ABB RobotStudio station: L4_1_20220629-155623.rsstn

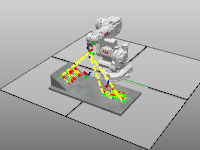
Station L4_1 (saved by RobotStudio 20.4.9280.0)
Controller IRB140_6_81
  mechanical unit ROB_1: IRB140_6_81_C_03, 6 joints, base frame (0, 0, 0) mm
Layout (positions relative to the parent item):
  - IRB140_6_81_C_03 [mechanism, from Robots\IRB140_6_81_C_G_03.rslib] at (0, 0, 0) mm; joint values [0, 0, 0, 0, 0.5236, 0] (rad or m)
  - MyNewTool [mechanism] at (506.29, 0, 679.5) mm, rotated rx 180 ry 60 rz 180 deg
      TCP Point at (78.44, 0, 73.52) mm, rotated rx 0 ry 70 rz 0 deg
      links: Tool
  - BaseBoard [part]
  - InclinedBoard [part] at (230, -500, 30) mm
Attachment: MyNewTool is attached to IRB140_6_81_C_03 / Link6
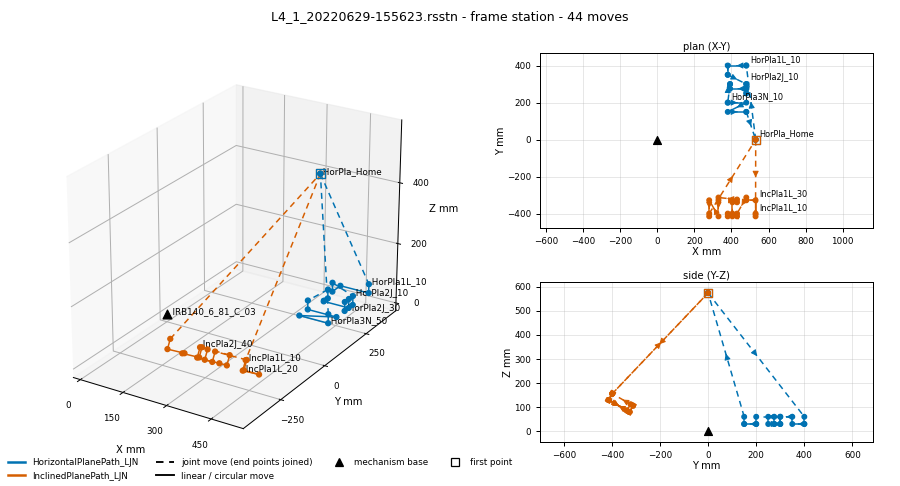
[picture p0: tool path of L4_1_20220629-155623.rsstn in frame station, 44 of 44 moves have a stored position in this frame; points joined in program order, loops and branches not executed]
Targets, tools, work objects and paths stored in the station, written as RAPID:
! task T_ROB1
MODULE CalibData
  TASK PERS wobjdata WO_InclinedPlane:=[FALSE,TRUE,"",[[230,-240.192,30],[0.68301276,-0.183012486,-0.183012486,-0.68301276]],[[0,0,30],[1,0,0,0]]];
  PERS tooldata Point:=[TRUE,[[78.437,0,73.516],[0.819152044,0,0.573576436,0]],[0.25,[0,0,1],[1,0,0,0],0,0,0]];
  TASK PERS wobjdata WO_HorizontalPlane:=[FALSE,TRUE,"",[[280,100,30],[1,0,0,0]],[[0,0,30],[1,0,0,0]]];
ENDMODULE

! task T_ROB1
MODULE Module1
  CONST robtarget HorPla2J_20:=[[200,200,-30],[0,0,1,0],[0,0,-1,1],[9E+09,9E+09,9E+09,9E+09,9E+09,9E+09]];
  CONST robtarget HorPla2J_10:=[[200,200,0],[0,0,1,0],[0,0,-1,1],[9E+09,9E+09,9E+09,9E+09,9E+09,9E+09]];
  CONST robtarget HorPla2J_30:=[[200,150,-30],[0,0,1,0],[0,0,-1,1],[9E+09,9E+09,9E+09,9E+09,9E+09,9E+09]];
  CONST robtarget HorPla2J_40:=[[200,150,0],[0,0,1,0],[0,0,-1,1],[9E+09,9E+09,9E+09,9E+09,9E+09,9E+09]];
  CONST robtarget HorPla2J_60:=[[200,175,-30],[0,0,1,0],[0,0,-1,1],[9E+09,9E+09,9E+09,9E+09,9E+09,9E+09]];
  CONST robtarget HorPla2J_50:=[[200,175,0],[0,0,1,0],[0,0,-1,1],[9E+09,9E+09,9E+09,9E+09,9E+09,9E+09]];
  CONST robtarget HorPla2J_70:=[[112.5,175,-30],[0,0,1,0],[0,0,-1,1],[9E+09,9E+09,9E+09,9E+09,9E+09,9E+09]];
  CONST robtarget HorPla2J_80:=[[100,187.5,-30],[0,0,1,0],[0,0,0,1],[9E+09,9E+09,9E+09,9E+09,9E+09,9E+09]];
  CONST robtarget HorPla2J_90:=[[112.5,200,-30],[0,0,1,0],[0,0,-1,1],[9E+09,9E+09,9E+09,9E+09,9E+09,9E+09]];
  CONST robtarget HorPla2J_100:=[[112.5,200,0],[0,0,1,0],[0,0,-1,1],[9E+09,9E+09,9E+09,9E+09,9E+09,9E+09]];
  CONST robtarget HorPla1L_10:=[[200,300,0],[0,0,1,0],[0,0,-1,1],[9E+09,9E+09,9E+09,9E+09,9E+09,9E+09]];
  CONST robtarget HorPla1L_30:=[[100,300,-30],[0,0,1,0],[0,0,-1,1],[9E+09,9E+09,9E+09,9E+09,9E+09,9E+09]];
  CONST robtarget HorPla1L_40:=[[100,250,-30],[0,0,1,0],[0,0,-1,1],[9E+09,9E+09,9E+09,9E+09,9E+09,9E+09]];
  CONST robtarget HorPla1L_50:=[[100,250,0],[0,0,1,0],[0,0,-1,1],[9E+09,9E+09,9E+09,9E+09,9E+09,9E+09]];
  CONST robtarget HorPla3N_20:=[[100,100,-30],[0,0,1,0],[0,0,0,1],[9E+09,9E+09,9E+09,9E+09,9E+09,9E+09]];
  CONST robtarget HorPla3N_10:=[[100,100,0],[0,0,1,0],[0,0,0,1],[9E+09,9E+09,9E+09,9E+09,9E+09,9E+09]];
  CONST robtarget HorPla3N_30:=[[200,100,-30],[0,0,1,0],[0,0,-1,1],[9E+09,9E+09,9E+09,9E+09,9E+09,9E+09]];
  CONST robtarget HorPla3N_40:=[[100,50,-30],[0,0,1,0],[0,0,0,1],[9E+09,9E+09,9E+09,9E+09,9E+09,9E+09]];
  CONST robtarget HorPla3N_50:=[[200,50,-30],[0,0,1,0],[0,0,-1,1],[9E+09,9E+09,9E+09,9E+09,9E+09,9E+09]];
  CONST robtarget HorPla1L_20:=[[200,300,-30],[0,0,1,0],[0,0,-1,1],[9E+09,9E+09,9E+09,9E+09,9E+09,9E+09]];
  CONST robtarget HorPla3N_60:=[[200,50,0],[0,0,1,0],[0,0,-1,1],[9E+09,9E+09,9E+09,9E+09,9E+09,9E+09]];
  CONST robtarget IncPla1L_10:=[[200,300,0],[0,0,1,0],[-1,0,-1,1],[9E+09,9E+09,9E+09,9E+09,9E+09,9E+09]];
  CONST robtarget IncPla1L_20:=[[200,300,-30],[0,0,1,0],[-1,0,-1,1],[9E+09,9E+09,9E+09,9E+09,9E+09,9E+09]];
  CONST robtarget IncPla1L_30:=[[100,300,-30],[0,0,1,0],[-1,0,-1,1],[9E+09,9E+09,9E+09,9E+09,9E+09,9E+09]];
  CONST robtarget IncPla1L_40:=[[100,250,-30],[0,0,1,0],[-1,0,-1,1],[9E+09,9E+09,9E+09,9E+09,9E+09,9E+09]];
  CONST robtarget IncPla1L_50:=[[100,250,0],[0,0,1,0],[-1,0,-1,1],[9E+09,9E+09,9E+09,9E+09,9E+09,9E+09]];
  CONST robtarget IncPla2J_10:=[[200,200,0],[0,0,1,0],[-1,0,-1,1],[9E+09,9E+09,9E+09,9E+09,9E+09,9E+09]];
  CONST robtarget IncPla2J_20:=[[200,200,-30],[0,0,1,0],[-1,0,-1,1],[9E+09,9E+09,9E+09,9E+09,9E+09,9E+09]];
  CONST robtarget IncPla2J_30:=[[200,150,-30],[0,0,1,0],[-1,0,-1,1],[9E+09,9E+09,9E+09,9E+09,9E+09,9E+09]];
  CONST robtarget IncPla2J_40:=[[200,150,0],[0,0,1,0],[-1,0,-1,1],[9E+09,9E+09,9E+09,9E+09,9E+09,9E+09]];
  CONST robtarget IncPla2J_50:=[[200,175,0],[0,0,1,0],[-1,0,-1,1],[9E+09,9E+09,9E+09,9E+09,9E+09,9E+09]];
  CONST robtarget IncPla2J_60:=[[200,175,-30],[0,0,1,0],[0,0,-1,1],[9E+09,9E+09,9E+09,9E+09,9E+09,9E+09]];
  CONST robtarget IncPla2J_70:=[[112.5,175,-30],[0,0,1,0],[-1,0,-1,1],[9E+09,9E+09,9E+09,9E+09,9E+09,9E+09]];
  CONST robtarget IncPla2J_80:=[[100,187.5,-30],[0,0,1,0],[-1,0,-1,1],[9E+09,9E+09,9E+09,9E+09,9E+09,9E+09]];
  CONST robtarget IncPla2J_90:=[[112.5,200,-30],[0,0,1,0],[-1,0,-1,1],[9E+09,9E+09,9E+09,9E+09,9E+09,9E+09]];
  CONST robtarget IncPla2J_100:=[[112.5,200,0],[0,0,1,0],[-1,0,-1,1],[9E+09,9E+09,9E+09,9E+09,9E+09,9E+09]];
  CONST robtarget IncPla3N_10:=[[100,100,0],[0,0,1,0],[-1,0,-1,1],[9E+09,9E+09,9E+09,9E+09,9E+09,9E+09]];
  CONST robtarget IncPla3N_20:=[[100,100,-30],[0,0,1,0],[-1,0,0,1],[9E+09,9E+09,9E+09,9E+09,9E+09,9E+09]];
  CONST robtarget IncPla3N_30:=[[200,100,-30],[0,0,1,0],[-1,0,-1,1],[9E+09,9E+09,9E+09,9E+09,9E+09,9E+09]];
  CONST robtarget IncPla3N_40:=[[100,50,-30],[0,0,1,0],[-1,0,0,1],[9E+09,9E+09,9E+09,9E+09,9E+09,9E+09]];
  CONST robtarget IncPla3N_50:=[[200,50,-30],[0,0,1,0],[-1,0,0,1],[9E+09,9E+09,9E+09,9E+09,9E+09,9E+09]];
  CONST robtarget IncPla3N_60:=[[200,50,0],[0,0,1,0],[0,0,-1,1],[9E+09,9E+09,9E+09,9E+09,9E+09,9E+09]];
  CONST robtarget HorPla_Home:=[[250.739874831,-100,514.813565403],[0.087155743,0,-0.996194698,0],[0,0,0,0],[9E+09,9E+09,9E+09,9E+09,9E+09,9E+09]];
  CONST robtarget IncPla_Home:=[[64.394019065,300.739878556,561.918401767],[0.241844546,0.696364278,-0.664463103,-0.122787591],[0,0,0,0],[9E+09,9E+09,9E+09,9E+09,9E+09,9E+09]];
  PROC main()
    HorizontalPlanePath_LJN;
    InclinedPlanePath_LJN;
  ENDPROC
  PROC HorizontalPlanePath_LJN()
    MoveJ HorPla_Home,v200,z10,Point\WObj:=WO_HorizontalPlane;
    MoveJ HorPla1L_10,v200,z10,Point\WObj:=WO_HorizontalPlane;
    MoveL HorPla1L_20,v100,z10,Point\WObj:=WO_HorizontalPlane;
    MoveL HorPla1L_30,v100,z10,Point\WObj:=WO_HorizontalPlane;
    MoveL HorPla1L_40,v100,z10,Point\WObj:=WO_HorizontalPlane;
    MoveL HorPla1L_50,v100,z10,Point\WObj:=WO_HorizontalPlane;
    MoveJ HorPla2J_10,v200,z10,Point\WObj:=WO_HorizontalPlane;
    MoveL HorPla2J_20,v100,z10,Point\WObj:=WO_HorizontalPlane;
    MoveL HorPla2J_30,v100,z10,Point\WObj:=WO_HorizontalPlane;
    MoveL HorPla2J_40,v100,z10,Point\WObj:=WO_HorizontalPlane;
    MoveJ HorPla2J_50,v200,z10,Point\WObj:=WO_HorizontalPlane;
    MoveL HorPla2J_60,v100,z10,Point\WObj:=WO_HorizontalPlane;
    MoveL HorPla2J_70,v100,z10,Point\WObj:=WO_HorizontalPlane;
    MoveC HorPla2J_80,HorPla2J_90,v100,z10,Point\WObj:=WO_HorizontalPlane;
    MoveL HorPla2J_100,v100,z10,Point\WObj:=WO_HorizontalPlane;
    MoveJ HorPla3N_10,v200,z10,Point\WObj:=WO_HorizontalPlane;
    MoveL HorPla3N_20,v100,z10,Point\WObj:=WO_HorizontalPlane;
    MoveL HorPla3N_30,v100,z10,Point\WObj:=WO_HorizontalPlane;
    MoveL HorPla3N_40,v100,z10,Point\WObj:=WO_HorizontalPlane;
    MoveL HorPla3N_50,v100,z10,Point\WObj:=WO_HorizontalPlane;
    MoveL HorPla3N_60,v100,z10,Point\WObj:=WO_HorizontalPlane;
    MoveJ HorPla_Home,v200,z10,Point\WObj:=WO_HorizontalPlane;
  ENDPROC
  PROC InclinedPlanePath_LJN()
    MoveJ IncPla_Home,v200,z10,Point\WObj:=WO_InclinedPlane;
    MoveJ IncPla1L_10,v200,z10,Point\WObj:=WO_InclinedPlane;
    MoveL IncPla1L_20,v100,z10,Point\WObj:=WO_InclinedPlane;
    MoveL IncPla1L_30,v100,z10,Point\WObj:=WO_InclinedPlane;
    MoveL IncPla1L_40,v100,z10,Point\WObj:=WO_InclinedPlane;
    MoveL IncPla1L_50,v100,z10,Point\WObj:=WO_InclinedPlane;
    MoveJ IncPla2J_10,v200,z10,Point\WObj:=WO_InclinedPlane;
    MoveL IncPla2J_20,v100,z10,Point\WObj:=WO_InclinedPlane;
    MoveL IncPla2J_30,v100,z10,Point\WObj:=WO_InclinedPlane;
    MoveL IncPla2J_40,v100,z10,Point\WObj:=WO_InclinedPlane;
    MoveJ IncPla2J_50,v200,z10,Point\WObj:=WO_InclinedPlane;
    MoveL IncPla2J_60,v100,z10,Point\WObj:=WO_InclinedPlane;
    MoveL IncPla2J_70,v100,z10,Point\WObj:=WO_InclinedPlane;
    MoveC IncPla2J_80,IncPla2J_90,v100,z10,Point\WObj:=WO_InclinedPlane;
    MoveL IncPla2J_100,v100,z10,Point\WObj:=WO_InclinedPlane;
    MoveJ IncPla3N_10,v200,z10,Point\WObj:=WO_InclinedPlane;
    MoveL IncPla3N_20,v100,z10,Point\WObj:=WO_InclinedPlane;
    MoveL IncPla3N_30,v100,z10,Point\WObj:=WO_InclinedPlane;
    MoveL IncPla3N_40,v100,z10,Point\WObj:=WO_InclinedPlane;
    MoveL IncPla3N_50,v100,z10,Point\WObj:=WO_InclinedPlane;
    MoveL IncPla3N_60,v100,z10,Point\WObj:=WO_InclinedPlane;
    MoveJ IncPla_Home,v200,z10,Point\WObj:=WO_InclinedPlane;
  ENDPROC
ENDMODULE

